// SIMATIC STEP 7 (V5.x) project RLI-p2
// CPU: CPU 412-1
// CPU: CPU 412-1
// station: Matériel
// station: Maitre
// station: Matériel
// station: Esclave
// station: P_ADR_BUS
// station: P_ADR_BUS
// program: Programme S7(1)
// program: Programme S7(2)

DATA_BLOCK DB 10
VERSION : 0.1
  STRUCT
   DB_VAR : INT  := 5;	//Variable temporaire de réservation
   VAR1 : INT  := 6;
   VAR2 : INT  := 7;
  END_STRUCT ;	
BEGIN
   DB_VAR := 5;
   VAR1 := 6;
   VAR2 := 7;
END_DATA_BLOCK

DATA_BLOCK DB 20
AUTHOR : SIMATIC
FAMILY : COM_FUNC
VERSION : 0.0
SFB 8
BEGIN
END_DATA_BLOCK

ORGANIZATION_BLOCK OB 1
TITLE = "Main Program Sweep (Cycle)"
VERSION : 0.1
VAR_TEMP
  OB1_EV_CLASS : BYTE ;	//Bits 0-3 = 1 (Coming event), Bits 4-7 = 1 (Event class 1)
  OB1_SCAN_1 : BYTE ;	//1 (Cold restart scan 1 of OB 1), 3 (Scan 2-n of OB 1)
  OB1_PRIORITY : BYTE ;	//Priority of OB Execution
  OB1_OB_NUMBR : BYTE ;	//1 (Organization block 1, OB1)
  OB1_RESERVED_1 : BYTE ;	//Reserved for system
  OB1_RESERVED_2 : BYTE ;	//Reserved for system
  OB1_PREV_CYCLE : INT ;	//Cycle time of previous OB1 scan (milliseconds)
  OB1_MIN_CYCLE : INT ;	//Minimum cycle time of OB1 (milliseconds)
  OB1_MAX_CYCLE : INT ;	//Maximum cycle time of OB1 (milliseconds)
  OB1_DATE_TIME : DATE_AND_TIME ;	//Date and time OB1 started
END_VAR
BEGIN
NETWORK
TITLE =
      A     I 0.0;
      =     L 20.0;
      BLD   103;
      BLD   9;
      =     L 25.0;
      CDB;
      OPN   DI 20;
      TAR2  LD 21;
      A     L 20.0;
      =     DIX 0.0;
      L     20;
      T     DIW 2;
      L     L#4;
      T     DID 4;
      L     W#16#1004;
      T     DIW 12;
      L     3;
      T     DIW 14;
      L     10;
      T     DIW 16;
      L     P#DBX 0.0;
      T     DID 18;
      LAR2  P#DBX 0.0;
      UC    SFB 8;
      LAR2  LD 21;
      A     DIX 8.1;
      =     Q 0.4;
      L     DIW 10;
      T     MW 20;
      CDB;
      BLD   10;
      NOP   0;
END_ORGANIZATION_BLOCK

SYMBOL_TABLE
"URCV"	SFB 9	SFB 9	// Uncoordinated Receiving of Data
END_SYMBOL_TABLE

DATA_BLOCK DB 11
VERSION : 0.1
  STRUCT
   DB_VAR : INT ;	//Variable temporaire de réservation
   var1 : INT ;
   VAr2 : INT ;
  END_STRUCT ;	
BEGIN
END_DATA_BLOCK

DATA_BLOCK DB 20
AUTHOR : SIMATIC
FAMILY : COM_FUNC
VERSION : 0.0
"URCV"
BEGIN
END_DATA_BLOCK

ORGANIZATION_BLOCK OB 1
TITLE = "Main Program Sweep (Cycle)"
VERSION : 0.1
VAR_TEMP
  OB1_EV_CLASS : BYTE ;	//Bits 0-3 = 1 (Coming event), Bits 4-7 = 1 (Event class 1)
  OB1_SCAN_1 : BYTE ;	//1 (Cold restart scan 1 of OB 1), 3 (Scan 2-n of OB 1)
  OB1_PRIORITY : BYTE ;	//Priority of OB Execution
  OB1_OB_NUMBR : BYTE ;	//1 (Organization block 1, OB1)
  OB1_RESERVED_1 : BYTE ;	//Reserved for system
  OB1_RESERVED_2 : BYTE ;	//Reserved for system
  OB1_PREV_CYCLE : INT ;	//Cycle time of previous OB1 scan (milliseconds)
  OB1_MIN_CYCLE : INT ;	//Minimum cycle time of OB1 (milliseconds)
  OB1_MAX_CYCLE : INT ;	//Maximum cycle time of OB1 (milliseconds)
  OB1_DATE_TIME : DATE_AND_TIME ;	//Date and time OB1 started
END_VAR
BEGIN
NETWORK
TITLE =
      A     I 0.0;
      =     L 20.0;
      BLD   103;
      BLD   9;
      =     L 25.0;
      CDB;
      OPN   DI 20;
      TAR2  LD 21;
      A     L 20.0;
      =     DIX 0.0;
      L     6;
      T     DIW 2;
      L     L#4;
      T     DID 4;
      L     W#16#1004;
      T     DIW 12;
      L     3;
      T     DIW 14;
      L     11;
      T     DIW 16;
      L     P#DBX 0.0;
      T     DID 18;
      LAR2  P#DBX 0.0;
      UC    "URCV";
      LAR2  LD 21;
      A     DIX 8.1;
      =     Q 0.4;
      L     DIW 10;
      T     MW 20;
      CDB;
      BLD   10;
      NOP   0;
END_ORGANIZATION_BLOCK
